Staubli VAL3: page_viewTraj.dtx

num nIndex
num nKey = 255
num nOldIndex = 2
public num nPage
num nRefresh = 13186.401
num nSelect
num nTime = 1
num nView
num nClockStatus
string sEvent = " 3. "
public string sItems = "test"
string sList[3]
  [0] = " 1. "
  [1] = " 2. "
  [2] = " 3. "
string sMenu[8]
  [0] = "Tool Selection"
  [2] = "Rename"
  [3] = "Paste"
  [4] = "Mark"
  [5] = "Delete"
  [6] = "Insert"
  [7] = "Save"
string sMenuUser[8]
string sMessage
string sTrajName = "test"
string sMenu8[8]
bool bButton[8]
  [0] = true
  [2] = true
  [3] = true
  [4] = true
  [5] = true
  [6] = true
  [7] = true
bool bLarge
bool bShowStatus
bool bExit
bool bTrigger
InstrItem iInstruction
  [0]
    string sType
    string sData
tool tTool = {fatherId=flange[0], ioLink=valve1}
frame fFather = {fatherId=world[0]}
num nBackupFrame
